(******************************************************************************
Baustein: FB_TestReportBase
Spezifikation: doc/Spezifikation.pdf, Kap. x.y.z
-------------------------------------------------------------------------------
erstellt:
von:
Geändert:
von:
-------------------------------------------------------------------------------
Beschreibung
Dieser Baustein enthält alle zugeordneten Testfälle. Ein Testfall
ist ein abgeleiteter Baustein (FB) von FB_UnitTestBase.

-------------------------------------------------------------------------------
Input
-

Output
-
******************************************************************************)
FUNCTION_BLOCK FB_FileBase
VAR_INPUT
END_VAR
VAR_OUTPUT
	o_bOpen 	: BOOL;
	o_bError 	: BOOL;
	o_bEmpty 	: BOOL;
END_VAR
VAR
	Buffer      : ARRAY[0..2048] OF BYTE;
	u32RdIdx    : UDINT;
	u32WrIdx    : UDINT;
	u32MaxIdx   : UDINT := 2048;
	
	fbOpen      : FB_FileOpen;
	fbClose     : FB_FileClose;
	fbWrite	    : FB_FileWrite;
	strFileName : StrFileName_t;
	strFilePath : StrPathName_t;
	
	eState 		: EExportState_t;
	u32Line     : UDINT;
	
	sStatistic  : SStatistic_t;

	trgOpen 	: F_TRIG;
	trgWrite 	: F_TRIG;
	trgClose 	: F_TRIG;
END_VAR


	fbOpen();
	fbWrite();
	fbClose();
	
	trgOpen(CLK := fbOpen.bBusy);
	IF trgOpen.Q = TRUE THEN
		fbOpen.bExecute := FALSE;
	END_IF;

	trgWrite(CLK := fbWrite.bBusy);
	IF trgWrite.Q = TRUE THEN
		fbWrite.bExecute := FALSE;
	END_IF;

	trgClose(CLK := fbClose.bBusy);
	IF trgClose.Q = TRUE THEN
		fbClose.bExecute := FALSE;
	END_IF;

	o_bEmpty := (u32WrIdx = u32RdIdx);

(******************************************************************************
Baustein: FB_TestReportBase.addCrlf
Spezifikation: doc/Spezifikation.pdf, Kap. x.y.z
-------------------------------------------------------------------------------
erstellt:
von:
Geändert:
von:
-------------------------------------------------------------------------------
Beschreibung


-------------------------------------------------------------------------------
Input
-

Output
-
******************************************************************************)
METHOD PUBLIC addCrlf : ERetCode_t
VAR_INPUT
END_VAR
VAR
	strTemp : string := '$R$N';
END_VAR

	addData(adr(strTemp), 2);
	
	addCrlf := ERetCode_t.eRetDone;
END_METHOD

METHOD PRIVATE addData : BOOL
VAR_INPUT
	pData   : POINTER TO BYTE;
	u32Size : UDINT;
END_VAR
VAR
	u32Part1 : UDINT;
	u32Part2 : UDINT;
END_VAR

	IF u32WrIdx + u32Size <= u32MaxIdx THEN
		MemCpy(ADR(buffer)+u32WrIdx, pData, u32Size);
		u32WrIdx := u32WrIdx + u32Size;
	ELSE
		// buffer bis maximum beschreiben und den rest
		// vorne einfügen
		u32Part1 := u32MaxIdx-u32WrIdx;
		u32Part2 := u32Size - u32Part1;

		MemCpy(ADR(buffer) + u32WrIdx, pData, u32Part1);
		
		MemCpy(ADR(buffer), pData+u32Part1, u32Part2);
		// Schreibindex ist dann die Restgröße in Byte
		u32WrIdx := u32Part2;
	END_IF
END_METHOD

(******************************************************************************
Baustein: FB_TestReportBase.addString
Spezifikation: doc/Spezifikation.pdf, Kap. x.y.z
-------------------------------------------------------------------------------
erstellt:
von:
Geändert:
von:
-------------------------------------------------------------------------------
Beschreibung

-------------------------------------------------------------------------------
Input
	i_strData : STRING(255);

Output
-
******************************************************************************)
METHOD PUBLIC addString : ERetCode_t
VAR_INPUT
	i_strData : STRING(255);
END_VAR

	addData(ADR(i_strData), len(i_strData));
	
	addString := ERetcode_t.eRetDone;
END_METHOD

METHOD PUBLIC addTimeMs : ERetCode_t
VAR_INPUT
	i_u32Value : UDINT;
END_VAR
VAR
	strTemp  : STRING;
	s16Len   : INT;
END_VAR


		strTemp := UDINT_TO_STRING(i_u32Value);
		s16Len  := len(strTemp);

		IF s16Len < 4 THEN

			WHILE s16Len < 3 DO
				strTemp := concat('0', strTemp);
				s16Len  := len(strTemp);
			END_WHILE

			strTemp := concat('.', strTemp);
			strTemp := concat('0', strTemp);

		END_IF;

		PRG_UnitTestLib.logInfo(concat('addTimeMs : ' , strTemp));

		addString(strTemp);
END_METHOD

(******************************************************************************
Baustein: FB_TestReportBase.addValue
Spezifikation: doc/Spezifikation.pdf, Kap. x.y.z
-------------------------------------------------------------------------------
erstellt:
von:
Geändert:
von:
-------------------------------------------------------------------------------
Beschreibung

-------------------------------------------------------------------------------
Input
	i_anyValue : ANY;

Output
-
******************************************************************************)
METHOD PUBLIC addValue : ERetCode_t
VAR_INPUT
	i_anyValue : ANY;
END_VAR
VAR
	uValue : UBaseTypes_t;
END_VAR

	addValue  := ERetcode_t.eRetDone;
	
	IF i_anyValue.pValue = 0 THEN
		addValue  := ERetcode_t.eRetFailed;
		RETURN;
	END_IF

	MEMCPY(ADR(uValue),i_anyValue.pValue, TO_UDINT(i_anyValue.diSize)); 

	CASE i_anyValue.TypeClass OF

	IBaseLibrary.TYPE_SINT:

		addString(SINT_TO_STRING(uValue.s8Value));

	IBaseLibrary.TYPE_USINT:

		addString(USINT_TO_STRING(uValue.u8Value));

	IBaseLibrary.TYPE_INT:

		addString(INT_TO_STRING(uValue.s16Value));

	IBaseLibrary.TYPE_DINT:

		addString(DINT_TO_STRING(uValue.s32Value));

	IBaseLibrary.TYPE_UINT:

		addString(UINT_TO_STRING(uValue.u16Value));

	IBaseLibrary.TYPE_UDINT:

		addString(UDINT_TO_STRING(uValue.u32Value));

	IBaseLibrary.TYPE_WORD:

		addString(WORD_TO_STRING(uValue.w16Value));

	IBaseLibrary.TYPE_DWORD:

		addString(DWORD_TO_STRING(uValue.w32Value));

	IBaseLibrary.TYPE_BYTE:

		addString(BYTE_TO_STRING(uValue.u8Value));

	IBaseLibrary.TYPE_BOOL:
		
		IF (uValue.bValue = TRUE) THEN
			addString('TRUE');
		ELSE
			addString('FALSE');
		END_IF;

	IBaseLibrary.TYPE_REAL:
		
		addString(REAL_TO_STRING(uValue.r32Value));
	
	ELSE
		ADSLOGSTR(msgCtrlMask 	:= ADSLOG_MSGTYPE_ERROR , 
				  msgFmtStr 	:= 'TestReportBase.AddValue: Unbekannter Datentyp!', 
				  strArg 		:= '');
	END_CASE;
END_METHOD

(******************************************************************************
Baustein: FB_TestReportBase.clearBuffer
Spezifikation: doc/Spezifikation.pdf, Kap. x.y.z
-------------------------------------------------------------------------------
erstellt:
von:
Geändert:
von:
-------------------------------------------------------------------------------
Beschreibung

-------------------------------------------------------------------------------
Input
-

Output
-
******************************************************************************)
METHOD PUBLIC clearBuffer : ERetCode_t
VAR_INPUT
END_VAR

	clearBuffer := ERetCode_t.eRetDone;
	
	MemSet(ADR(buffer), 0, SIZEOF(buffer));
	
	u32WrIdx := u32RdIdx := 0;
END_METHOD

(******************************************************************************
Baustein: FB_TestReportBase.Close
Spezifikation: doc/Spezifikation.pdf, Kap. x.y.z
-------------------------------------------------------------------------------
erstellt:
von:
Geändert:
von:
-------------------------------------------------------------------------------
Beschreibung


-------------------------------------------------------------------------------
Input
-

Output
-
******************************************************************************)
METHOD PUBLIC Close : ERetCode_t
VAR_INPUT
END_VAR

	Close := ERetCode_t.eRetBusy;
	
	fbClose.hFile 		:= fbOpen.hFile;

	IF o_bEmpty = TRUE THEN

		fbClose.bExecute 	:= TRUE; 

		IF trgClose.Q = TRUE THEN
			o_bOpen 			:= FALSE;
		END_IF;	
		
		IF fbClose.bError = TRUE THEN
			Close := eRetCode_t.eRetFailed;
		END_IF;			

	END_IF;

	IF o_bOpen = FALSE THEN
		Close 				:= ERetCode_t.eRetDone;
		fbClose.bExecute 	:= FALSE;		
	END_IF;
END_METHOD

(******************************************************************************
Baustein: FB_TestReportBase.getFileName
Spezifikation: doc/Spezifikation.pdf, Kap. x.y.z
-------------------------------------------------------------------------------
erstellt:
von:
Geändert:
von:
-------------------------------------------------------------------------------
Beschreibung
Diese Methode muss vom ableitenden Baustein überschrieben werden und
wird von der Basisklasse aus aufgerufen wenn der Report erstellt werden
soll.

-------------------------------------------------------------------------------
Input
	i_pFileName : NameHandle_t;
	i_pPath		: PathHandle_t;

Output
-
******************************************************************************)
METHOD PROTECTED getFileName : ERetCode_t
VAR_INPUT
	i_pFileName : NameHandle_t;
	i_pPath		: PathHandle_t;
END_VAR
END_METHOD

(******************************************************************************
Baustein: FB_TestReportBase.getTime
Spezifikation: doc/Spezifikation.pdf, Kap. x.y.z
-------------------------------------------------------------------------------
erstellt:
von:
Geändert:
von:
-------------------------------------------------------------------------------
Beschreibung


-------------------------------------------------------------------------------
Input
-

Output
-
******************************************************************************)
METHOD PROTECTED getTime : TimeStruct
VAR_INPUT
END_VAR
VAR
END_VAR

	getTime := PRG_UnitTestLib.getTime();
END_METHOD

(******************************************************************************
Baustein: FB_TestReportBase.Open
Spezifikation: doc/Spezifikation.pdf, Kap. x.y.z
-------------------------------------------------------------------------------
erstellt:
von:
Geändert:
von:
-------------------------------------------------------------------------------
Beschreibung


-------------------------------------------------------------------------------
Input
-

Output
-
******************************************************************************)
METHOD PUBLIC open : ERetCode_t
VAR_INPUT
	i_strPath : StrPathName_t;
	i_strName : StrFileName_t;
END_VAR

	open := ERetCode_t.eRetBusy;
	
	strFileName := i_strName;
	strFilePath := i_strPath;

	fbOpen.sPathName := CONCAT(strFilePath, strFileName);
	fbOpen.nMode 	 := FOPEN_MODEWRITE OR FOPEN_MODEBINARY;	
	fbOpen.bExecute  := TRUE;
			
	IF trgOpen.Q = TRUE THEN
		o_bOpen := true;
		fbOpen.bExecute  := FALSE;		
	END_IF;	
	
	IF fbOpen.bError = TRUE THEN
		open := eRetCode_t.eRetFailed;
	END_IF;	

	IF o_bOpen = TRUE THEN
		open := eRetCode_t.eRetDone;
	END_IF;
END_METHOD

(******************************************************************************
Baustein: FB_TestReportBase.reset
Spezifikation: doc/Spezifikation.pdf, Kap. x.y.z
-------------------------------------------------------------------------------
erstellt:
von:
Geändert:
von:
-------------------------------------------------------------------------------
Beschreibung


-------------------------------------------------------------------------------
Input
-

Output
-
******************************************************************************)
METHOD PUBLIC reset : BOOL
VAR_INPUT
END_VAR

	IF fbOpen.hFile <> 0 THEN
		close();
	END_IF
	
	clearBuffer();

	fbOpen(sPathName := '', bExecute := FALSE);
	
	fbWrite(bExecute := FALSE);
	
	fbClose(bExecute := FALSE);
	
	o_bOpen := false;
END_METHOD

(******************************************************************************
Baustein: FB_TestReportBase.writeBuffer
Spezifikation: doc/Spezifikation.pdf, Kap. x.y.z
-------------------------------------------------------------------------------
erstellt:
von:
Geändert:
von:
-------------------------------------------------------------------------------
Beschreibung


-------------------------------------------------------------------------------
Input
-

Output
-
******************************************************************************)
METHOD PUBLIC writeBuffer : ERetCode_t
VAR_INPUT
END_VAR
VAR
	u32Len : UDINT;
END_VAR

	writeBuffer := eRetCode_t.eRetBusy;

	IF fbWrite.bBusy = TRUE THEN
		RETURN;	
	ELSIF u32WrIdx = u32RdIdx THEN
		writeBuffer := eRetCode_t.eRetDone;
		RETURN;	
	END_IF
	
	IF u32WrIdx > u32RdIdx THEN
		u32Len := u32WrIdx - u32RdIdx; 
		writeBuffer := writeData(i_pData := ADR(Buffer)+u32RdIdx, u32Size := u32Len);	
	ELSE
		u32Len := u32MaxIdx - u32RdIdx; 
		writeBuffer := writeData(i_pData := ADR(Buffer)+ u32RdIdx, u32Size := u32Len);
		writeBuffer := writeData(i_pData := ADR(Buffer), u32Size := u32WrIdx);	
	END_IF;
END_METHOD

(******************************************************************************
Baustein: FB_TestReportBase.writeData
Spezifikation: doc/Spezifikation.pdf, Kap. x.y.z
-------------------------------------------------------------------------------
erstellt:
von:
Geändert:
von:
-------------------------------------------------------------------------------
Beschreibung


-------------------------------------------------------------------------------
Input
	i_pData : POINTER TO BYTE;
	u32Size : UDINT;
	
Output
-
******************************************************************************)
METHOD PROTECTED writeData : ERetCode_t
VAR_INPUT
	i_pData : POINTER TO BYTE;
	u32Size : UDINT;
END_VAR

	writeData := ERetCode_t.eRetFailed;
	
	IF u32Size = 0 OR i_pData = 0 THEN
		RETURN;
	END_IF
	
	fbWrite.pWriteBuff 	:= i_pData; 
	fbWrite.cbWriteLen 	:= u32Size; 
	fbWrite.hFile 		:= fbOpen.hFile; 

	fbWrite(bExecute 	:= TRUE);
			
	IF fbWrite.bBusy = FALSE THEN
		fbWrite(bExecute 	:= FALSE);	
		writeData 	:= ERetCode_t.eRetDone;
		u32RdIdx 	:= u32WrIdx;
	ELSE	
		writeData := ERetCode_t.eRetBusy;
	END_IF;	

	IF fbWrite.bError = TRUE THEN
		writeData := eRetCode_t.eRetFailed;
	END_IF;
END_METHOD

END_FUNCTION_BLOCK

(* stored: Version 1.1.0.1, ProductVersion 3.1.4024.3
   POU FB_FileBase: Id {ae4044ad-0900-4102-9c63-f2ca7dc7882b}, SpecialFunc None
   Method addCrlf: Id {87e751ae-43bf-42cc-9a5b-1406edf6821d}
   Method addData: Id {dc5bbd79-131e-449c-8aa9-a21e0c029bdd}
   Method addString: Id {9ba3d4d4-f543-4168-92a3-a04eafe3c218}
   Method addTimeMs: Id {09890850-d355-4c09-a6ca-8b26f87f9775}
   Method addValue: Id {4763b747-b35d-40cf-ae56-8465970254b3}
   Method clearBuffer: Id {5dfaa680-7bea-4746-bf0e-4660536af9df}
   Method Close: Id {03c998bc-5bf6-4151-a33b-ec883349b294}
   Method getFileName: Id {7e1d2ee9-2256-4e5a-8158-937367f08b2c}
   Method getTime: Id {d393fabf-7345-423a-9e35-8e600869be1d}
   Method open: Id {902b4c08-29bc-4d3a-8f22-681df2d06abd}
   Method reset: Id {e1e2a994-d63a-4204-a9c4-0718d80f0ccf}
   Method writeBuffer: Id {ffe30870-323c-4ba5-b165-beb9ce4f98c7}
   Method writeData: Id {8feaea14-66b2-4bf1-abf3-f924d7301621} *)
